// Mitsubishi GX Works2 project: 0709downcount   PLC: Q02/Q02H

PROGRAM MAIN
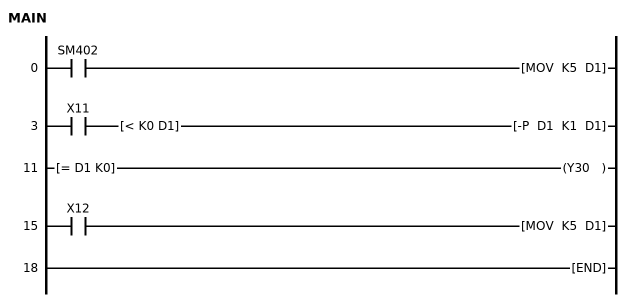
0     LD      SM402
      MOV     K5 D1
3     LD      X11
      AND<    K0 D1
      -P      D1 K1 D1
11    LD=     D1 K0
      OUT     Y30
15    LD      X12
      MOV     K5 D1
18    END
END_PROGRAM
